(* PLC project Tc2_Utilities.LcomplexIsNaN Demo, tc3-libraries-kb TwinCAT 3.1 *)
(* stored: creationDateTime 2026-05-10T11:00:00, modificationDateTime 2026-05-10T11:00:00 *)

PROGRAM P_Demo_LcomplexIsNaN
  VAR
    bResult : BOOL;  (* LcomplexIsNaN 的返回值 *)
    bRun : BOOL;  (* 触发一次调用 *)
    lcZ : LCOMPLEX;  (* 测试用本地变量 *)
  END_VAR

            // ============================================================
// Tc2_Utilities.LcomplexIsNaN 演示程序（FUNCTION）
// ============================================================
// 验证步骤：
//   1. 引用 Tc2_Utilities（及依赖类型所在的库）
//   2. 编译 + 登录
//   3. 强制 bRun := TRUE 一个周期
//   4. 观察 bResult 应为 FALSE（正常值）
// ============================================================

// 不赋 NaN 时 IsNaN = FALSE；可手动写 lcZ.r := 0.0/0.0; 测 TRUE
IF bRun THEN
    bResult := LcomplexIsNaN(lcZ);
    bRun := FALSE;
END_IF;

          
END_PROGRAM
